(* PLC project aaaa, Dassault Systèmes ControlBuild 2024x Refresh1 *)
(* stored: creationDateTime 2024-04-02T17:37:35-01:00 *)

PROGRAM aaaa.aaaa

(* FBD diagram, written out as Structured Text *)
END_PROGRAM
